Staubli VAL3: TRACK.pjx

--- TRACK.pjx ---
Parameters version=s7.8.3 stackSize=5000 millimeterUnit=true
Program file=copy_it.pgx
Program file=link_all.pgx
Program file=link_it.pgx
Program file=setMobile.pgx
Data file=TRACK.dtx
Library alias=saveData path=Disk://saveData/savedata.pjx
Type name=FrameItem path=Disk://kernel/template/FrameItem/FrameItem.pjx

--- TRACK.dtx ---
public Tracks tTraj{}

--- link_it.pgx ---
public program link_it(string x_sName)
begin
  // link all the point
  call link_all(x_sName)
end

--- setMobile.pgx ---
public program setMobile(string x_sItem, frame x_fFrame)
begin
  // set the frame mobile
  tTraj[x_sItem].fMoving.trsf={0,0,0,0,0,0}
  link(tTraj[x_sItem].fMoving,x_fFrame)
end
